Omron CX-Programmer project NewProject (CX-Programmer 9.70)

# PLC NewPLC1: CPM1(CPM1A) CPU20

## Global symbols (name address type ; comment)
0.00 BOOL  ; ON
0.01 BOOL  ; LLS4
0.02 BOOL  ; LLS1
0.03 BOOL  ; HLS1
0.04 BOOL  ; VS3
0.05 BOOL  ; FimCurso
0.06 BOOL  ; HLS4
0.07 BOOL  ; RESET
10.00 BOOL  ; Bomba
10.01 BOOL  ; VS1
10.02 BOOL  ; VS3
10.03 BOOL  ; LED LARANJA
10.04 BOOL  ; led verde
10.08 BOOL  ; VS3
10.09 BOOL  ; LED AZUL
200.01 BOOL  ; Intermitente
TIM001 BOOL  ; 5 Segundos

## Program NewProgram1 (no task)

### Section Section1

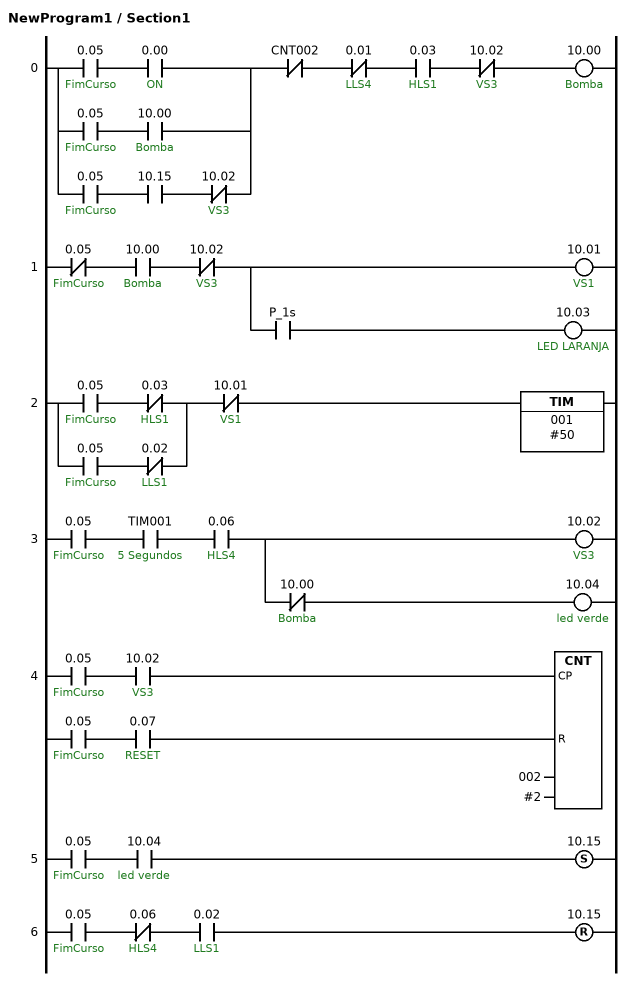
; rung 0
LD 0.05  ; FimCurso
AND 0.00  ; ON
LD 0.05  ; FimCurso
AND 10.00  ; Bomba
ORLD
LD 0.05  ; FimCurso
AND 10.15
ANDNOT 10.02  ; VS3
ORLD
ANDNOT CNT002
ANDNOT 0.01  ; LLS4
AND 0.03  ; HLS1
ANDNOT 10.02  ; VS3
OUT 10.00  ; Bomba
; rung 1
LDNOT 0.05  ; FimCurso
AND 10.00  ; Bomba
ANDNOT 10.02  ; VS3
OUT 10.01  ; VS1
AND P_1s
OUT 10.03  ; LED LARANJA
; rung 2
LD 0.05  ; FimCurso
ANDNOT 0.03  ; HLS1
LD 0.05  ; FimCurso
ANDNOT 0.02  ; LLS1
ORLD
ANDNOT 10.01  ; VS1
TIM 001 #50
; rung 3
LD 0.05  ; FimCurso
AND TIM001  ; 5 Segundos
AND 0.06  ; HLS4
OUT 10.02  ; VS3
ANDNOT 10.00  ; Bomba
OUT 10.04  ; led verde
; rung 4
LD 0.05  ; FimCurso
AND 10.02  ; VS3
LD 0.05  ; FimCurso
AND 0.07  ; RESET
CNT 002 #2
; rung 5
LD 0.05  ; FimCurso
AND 10.04  ; led verde
SET 10.15
; rung 6
LD 0.05  ; FimCurso
ANDNOT 0.06  ; HLS4
AND 0.02  ; LLS1
RSET 10.15

### Section END
; rung 0
END(01)